// TIA Portal V18 export
VAR_GLOBAL   // PLC tag table "PartType"
END_VAR
VAR_GLOBAL CONSTANT   // user constants
   PartTypeFor_11KW : USInt := 1;
   PartTypeFor_22KW : USInt := 2;
   Cy10GoHome : UInt := 0;
   Cy10GoWork : UInt := 1;
END_VAR
